VAR_GLOBAL
	IOUT_WD_RANGE	:	INT		:=32767;
	VOUT_WD_RANGE	:	INT		:=32767;
	
	A_FLOW_MAX 		:	LREAL	:=10.0;
	D_FLOW_MAX		:	LREAL	:=10000.0;
	E_FLOW_MAX		:	LREAL	:=10000.0;
	P_REACTOR_MAX	:	LREAL	:=3000.0;
	
	A_FLOW_MIN 		:	LREAL	:=0.0;
	D_FLOW_MIN		:	LREAL	:=0.0;
	E_FLOW_MIN		:	LREAL	:=0.0;
	P_REACTOR_MIN	:	LREAL	:=0.0;
	
	AOUT_MAX		:	LREAL	:=10.0;
	AOUT_MIN		:	LREAL	:=0.0;
END_VAR

(* stored: Version 1.1.0.1, ProductVersion 3.1.0.36
   GVL G_PARAMS: Id {3b9a06b5-e024-4474-8f53-bae8a479db56} *)
